{attribute addProperty BoxType "AT2050-0500-0024"}
{attribute addProperty Id "A_0089_AT2050_5501_0018_AT2050_5501AT2050_C5E5984862678.25"}
{attribute addProperty CRC "4141398732"}
{attribute addProperty SizeInBites "626"}
{attribute addProperty SizeInBytes "78.25"}
TYPE A_0055_AT2050_0500_0024_F6D8BACC EXTENDS AT2050_BA5A9548 :
STRUCT
	{attribute addProperty Name "A_0089_AT2050_5501_0018_AT2050_5501"}
	A_0089_AT2050_5501_0018_AT2050_5501 : AT2050_C5E59848;
END_STRUCT
END_TYPE

(* stored: Version 1.2.0.0, ProductVersion 3.1.4024.9
   DUT A_0055_AT2050_0500_0024_F6D8BACC: Id {82410a22-df7d-42d6-a0b4-bb52a7391fdf} *)
